(* Logix 5000 project; controller VentiladorCamaraFriaParte1 vendor 1 type 14 code 89 rev 20.12; software revision 20.04 *)

TASK MainTask (continuous, watchdog 500 ms) : MainProgram

MODULES
   Controller : vendor 1 type 14 code 89 (CompactLogixL23E_QBFC1_Controller 0, rev 20.12)
      LocalENB : vendor 1 type 12 code 191 (CompactLogixL23E_QBFC1_Ethernet 1, rev 20.11)
         Ventilador : vendor 1 type 127 code 40 (Ethernet 192.168.1.53, rev 6.2, Output RPI 20 ms)
             : vendor 1 type 127 code 33792 (DSI 1, rev 1.7)
      Local : CompactBus (CompactVirtualAdapter 3, rev 20.11)
         Discrete_Inputs : vendor 1 type 7 code 320 (Compact 1, rev 3.1, Input RPI 20 ms)
         Discrete_Outputs : vendor 1 type 7 code 322 (Compact 2, rev 3.1, Output RPI 20 ms)
         Analog_IO : vendor 1 type 10 code 120 (Compact 3, rev 1.1, Output RPI 80 ms)
         Counters : vendor 1 type 109 code 70 (Compact 4, rev 1.1, Output RPI 20 ms)
END_MODULES

VAR_GLOBAL   (* controller tags *)
   BSAdd : BOOL;
   Decrementa : BOOL;
   Incrementa : BOOL;
END_VAR

PROGRAM MainProgram   (* main routine MainRoutine *)
VAR
   AcionaMotor : BOOL;
   AddTempoLig : ALIAS FOR Local:1:I.Data.6;
   BDMotor : BOOL;
   BSStartInversor : BOOL;
   Conta : COUNTER := (PRE := 10);
   ContaLigado : COUNTER;
   DecTempoLig : ALIAS FOR Local:1:I.Data.7;
   Desliga : ALIAS FOR Local:1:I.Data.0;
   Desligou : BOOL;
   Liga : ALIAS FOR Local:1:I.Data.5;
   MaquinaLigada : BOOL;
   Motor : ALIAS FOR Local:2:O.Data.1;
   SinalTempoMax : ALIAS FOR Local:2:O.Data.2;
   SinalTempoMin : ALIAS FOR Local:2:O.Data.3;
   SobrecargaInversor : ALIAS FOR Local:1:I.Data.2;
   StartInversor : BOOL;
   StopInversor : BOOL;
   TempoDesligado : TIMER := (PRE := 8000);
   TempoLigado : TIMER := (PRE := 5000);
   teste : COUNTER;
END_VAR

ROUTINE MainRoutine   (* ladder *)
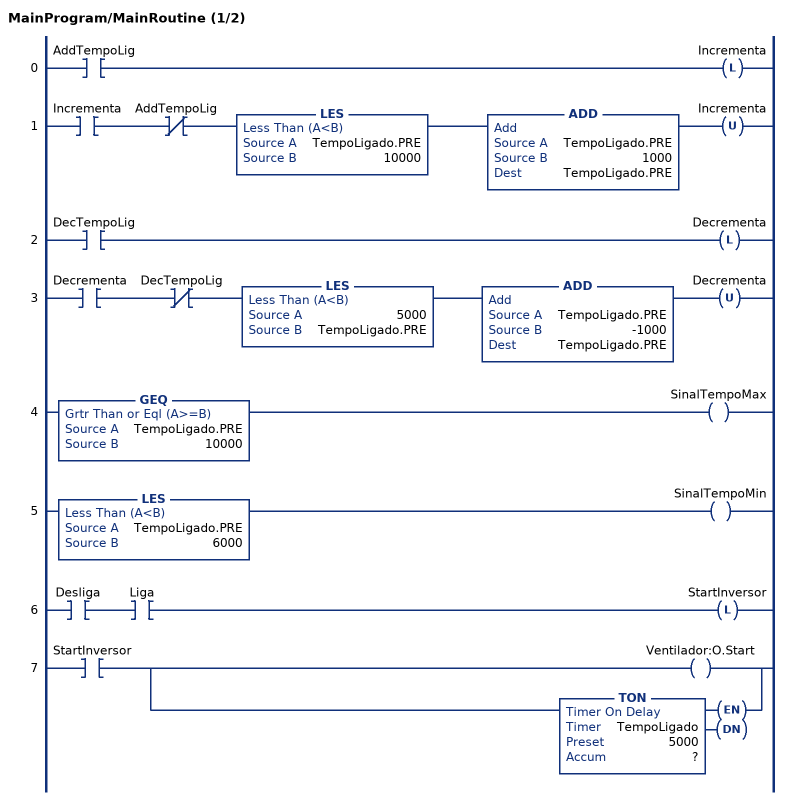
   0: XIC(AddTempoLig)OTL(Incrementa);
   1: XIC(Incrementa)XIO(AddTempoLig)LES(TempoLigado.PRE,10000)ADD(TempoLigado.PRE,1000,TempoLigado.PRE)OTU(Incrementa);
   2: XIC(DecTempoLig)OTL(Decrementa);
   3: XIC(Decrementa)XIO(DecTempoLig)LES(5000,TempoLigado.PRE)ADD(TempoLigado.PRE,-1000,TempoLigado.PRE)OTU(Decrementa);
   4: GEQ(TempoLigado.PRE,10000)OTE(SinalTempoMax);
   5: LES(TempoLigado.PRE,6000)OTE(SinalTempoMin);
   6: XIC(Desliga)XIC(Liga)OTL(StartInversor);
   7: XIC(StartInversor)[OTE(Ventilador:O.Start) ,TON(TempoLigado,?,?) ];
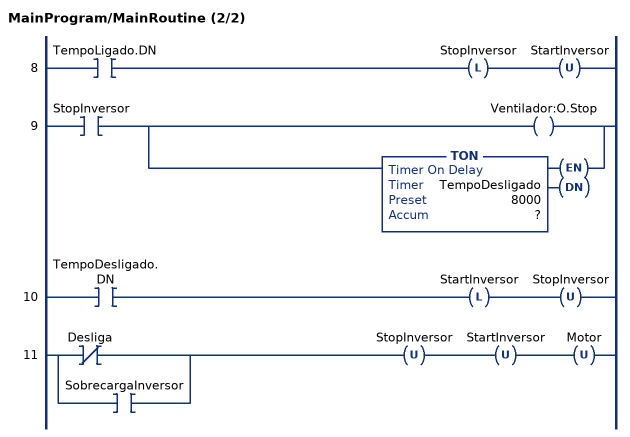
   8: XIC(TempoLigado.DN)OTL(StopInversor)OTU(StartInversor);
   9: XIC(StopInversor)[OTE(Ventilador:O.Stop) ,TON(TempoDesligado,?,?) ];
   10: XIC(TempoDesligado.DN)OTL(StartInversor)OTU(StopInversor);
   11: [XIO(Desliga) ,XIC(SobrecargaInversor) ]OTU(StopInversor)OTU(StartInversor)OTU(Motor);
END_ROUTINE
END_PROGRAM
